KUKA KRL program: EVEN.src

&ACCESS RV
&REL 1
&PARAM TEMPLATE = C:\KRC\Roboter\Template\FunctionVorgabe
&PARAM EDITMASK = *
DEFFCT BOOL EVEN(VALUE:IN )
  INT VALUE
  REAL VAL
  BOOL RET_VAL

  VAL = VALUE / 2.0
  RET_VAL = (DECIMAL(VAL) < 0.1)

  RETURN(RET_VAL)
ENDFCT
